(* Reference laser with X/Y motors (REFT): thin ND-framework state-mover
   wrapper. In/out mover via FB_PositionStatePMPSND, plus a tick site for
   the laser power/dimmer (FB_REF_Laser) and the X/Y motors. Caller-owned
   axes, stage/state arrays, fast-fault and arbiter injected via FB_Init
   REFERENCE TO and forwarded to fbStates; toggles re-forwarded each cycle. *)
{attribute 'call_after_init'}
FUNCTION_BLOCK FB_REFT
VAR_INPUT
    (* Device-specific state-enum bridges. Typed as E_EpicsInOut (UINT
       base) so the caller surface is enum-checked; the inline-init
       below binds them to FB_PositionStatePMPSND's REFERENCE TO UINT
       params via the shared UINT base. Callers drive moves with
       `fbREF.eEnumSet := E_EpicsInOut.OUT;` and read
       `fbREF.eEnumGet`. *)
    // Set this to a non-unknown value to request a new move.
    {attribute 'pytmc' := '
        pv: MMS:STATE:SET
        io: io
    '}
    eEnumSet : E_EpicsInOut;
    (* Run-time toggles forwarded into fbStates each cycle. PMPSND
       captures these by value in its own FB_Init, so the body
       re-writes fbStates.* every cycle to track live caller changes. *)
    fTermMax               : LREAL := 200;
END_VAR
VAR


    {attribute 'pytmc' := 'pv: LAS'}
    fbLaser : FB_REF_Laser;

    axisRefX : REFERENCE TO AXIS_REF;
    axisREFY : REFERENCE TO AXIS_REF;
     {attribute 'pytmc' := '
        pv: TST:Y
        io: io
        axis-link:
    '}
    fbMotorX : FB_MotionStageNC(
        AxisRef := axisRefX,
        iPersistentDataStorage := iPersistentDataStorage,
        sName := 'X'
    );
     {attribute 'pytmc' := '
        pv: TST:Y
        io: io
        axis-link:
    '}
    fbMotorY : FB_MotionStageNC(
        AxisRef := axisREFY,
        iPersistentDataStorage := iPersistentDataStorage,
        sName := 'Y'
    );

    iPersistentDataStorage : LCLS_Tc_DevAbs.I_PersistentDataStorage;
    aiMotionStage : ARRAY[1..MotionConstants.MAX_STATE_MOTORS] OF I_MotionStage := [fbMotorX, fbMotorY];

    astPositionState : REFERENCE TO ARRAY[1..MotionConstants.MAX_STATE_MOTORS]
                         OF ARRAY[1..GeneralConstants.MAX_STATES] OF ST_PositionState;

    {attribute 'no_copy'}
    fbFFHWO               : REFERENCE TO FB_HardwareFFOutput;
    {attribute 'no_copy'}
    fbArbiter             : REFERENCE TO FB_Arbiter;

    sDeviceName           : STRING;
    sTransitionKey        : STRING;
    bEnableMotion         : BOOL := TRUE;
    bEnableBeamParams     : BOOL;
    bEnablePositionLimits : BOOL;
    bReadDBNow            : BOOL;

    bFileReaderBusy       : REFERENCE TO BOOL;
    bFileReaderError      : REFERENCE TO BOOL;
    (* One configurator per REF state (OUT, IN). Writes the per-state
       sName and fDelta. Ticked cyclically in the body AFTER fbStates
       so its writes win over the template baseline FB_StateSetup
       applied via FB_CC_StatePMPSConfig *)
    afbStateDefaults : ARRAY[1..2] OF FB_CC_DeviceStateDefaults[
        (stPositionState := astPositionState[1][E_EpicsInOut.OUT],
         sName           := 'OUT',
         fDelta          := FDELTA_DEFAULT),
        (stPositionState := astPositionState[1][E_EpicsInOut.IN],
         sName           := 'IN',
         fDelta          := FDELTA_DEFAULT)
    ];
    {attribute 'pytmc' := 'pv: MMS'}
    fbStates : FB_PositionStatePMPSND(
        aiMotionStage         := aiMotionStage,
        astPositionState      := astPositionState,
        nActiveMotorCount     := 1,
        eEnumSet              := eEnumSet,
        eEnumGet              := eEnumGet,
        bEnableMotion         := bEnableMotion,
        eMotionRequestPolicy  := E_MotionRequestPolicy.INTERRUPT,
        bEnableBeamParams     := bEnableBeamParams,
        bEnablePositionLimits := bEnablePositionLimits,
        bReadDBNow            := bReadDBNow,
        bFileReaderBusy       := bFileReaderBusy,
        bFileReaderError      := bFileReaderError,
        fbFFHWO               := fbFFHWO,
        fbArbiter             := fbArbiter,
        sDeviceName           := sDeviceName,
        sTransitionKey        := sTransitionKey
    );
    i : UINT;
    bFirstScan: BOOL := TRUE;
END_VAR
VAR_OUTPUT
    // The current position state as an enum.
    {attribute 'pytmc' := '
        pv: MMS:STATE:GET
        io: i
    '}
     eEnumGet : E_EpicsInOut;
    // The PMPS database lookup associated with the current position state.
    stDbStateParams: ST_DbStateParams;
END_VAR
VAR CONSTANT
    (* REF-wide default tolerance for state in-position detection,
       applied per-state by afbStateDefaults. *)
    FDELTA_DEFAULT : LREAL := 2;
END_VAR

IF NOT __ISVALIDREF(astPositionState)
   OR NOT __ISVALIDREF(fbFFHWO)
   OR NOT __ISVALIDREF(fbArbiter) THEN
    RETURN;
END_IF

IF bFirstScan THEN
    FOR i := 1 TO MotionConstants.MAX_STATE_MOTORS DO
        aiMotionStage[i].SetModeEnableLimits(
            LimBackward    := TRUE,
            LimForward     := TRUE,
            HomeEnable     := FALSE,
            BrakeMode      := E_StageBrakeMode.IF_ENABLED,
            EnableMode     := E_StageEnableMode.DURING_MOTION,
            HomeMode       := E_EpicsHomeCmd.LOW_LIMIT,
            UserEnable     := TRUE,
            HardwareEnable := TRUE
        );
        aiMotionStage[i].SetVelocity(Velocity:=15.5);
        aiMotionStage[i].RestoreMotionParams:= FALSE;
    END_FOR
    bFirstScan := FALSE;
END_IF

fbStates(stDbStateParams=> stDbStateParams);

fbLaser(fTermMax := fTermMax);

fbMotorY();
fbMotorX();

(* Auto-fired after FB_Init. fbStates' inline-init ran first and
   forwarded nil refs, so this re-supplies the now-valid refs via
   fbStates.CallAfterInitStateMover / CallAfterInitPMPS and writes the
   per-state device defaults. *)
{attribute 'call_after_init'}
METHOD CallAfterInit
VAR
    i : UINT;
END_VAR
afbStateDefaults[1].CallAfterInit(
    stPositionState := THIS^.astPositionState[1][E_EpicsInOut.OUT]
);
afbStateDefaults[2].CallAfterInit(
    stPositionState := THIS^.astPositionState[1][E_EpicsInOut.IN]
);

THIS^.fbStates.CallAfterInitStateMover(
    aiMotionStage         := aiMotionStage,
    astPositionState      := astPositionState,
    nActiveMotorCount     := 1,
    eEnumSet              := eEnumSet,
    eEnumGet              := eEnumGet,
    bEnableMotion         := bEnableMotion,
    eMotionRequestPolicy  := E_MotionRequestPolicy.INTERRUPT,
);

THIS^.fbStates.CallAfterInitPMPS(
    aiMotionStage         := aiMotionStage,
    astPositionState      := astPositionState,
    bEnableBeamParams     := bEnableBeamParams,
    bEnablePositionLimits := bEnablePositionLimits,
    bReadDBNow            := bReadDBNow,
    bFileReaderBusy       := bFileReaderBusy,
    bFileReaderError      := bFileReaderError,
    fbFFHWO               := fbFFHWO,
    fbArbiter             := fbArbiter,
    sDeviceName           := sDeviceName,
    sTransitionKey        := sTransitionKey
);
END_METHOD

//FB_Init is always available implicitly and it is used primarily for initialization.
//The return value is not evaluated. For a specific influence, you can also declare the
//methods explicitly and provide additional code there with the standard initialization
//code. You can evaluate the return value.
METHOD FB_Init: BOOL
VAR_INPUT
    bInitRetains: BOOL; // TRUE: the retain variables are initialized (reset warm / reset cold)
    bInCopyCode: BOOL;  // TRUE: the instance will be copied to the copy code afterward (online change)
    astPositionState       : REFERENCE TO ARRAY[1..MotionConstants.MAX_STATE_MOTORS]
                                            OF ARRAY[1..GeneralConstants.MAX_STATES] OF ST_PositionState;
    axisRefX : REFERENCE TO AXIS_REF;
    axisREFY : REFERENCE TO AXIS_REF;
    fbFFHWO                : REFERENCE TO FB_HardwareFFOutput;
    fbArbiter              : REFERENCE TO FB_Arbiter;
    sDeviceName            : STRING;
    sTransitionKey         : STRING;
    bEnableBeamParams      : BOOL;
    bEnablePositionLimits  : BOOL;
    bReadDBNow             : BOOL;
    bFileReaderBusy       : REFERENCE TO BOOL;
    bFileReaderError      : REFERENCE TO BOOL;
END_VAR
THIS^.astPositionState REF= astPositionState;
THIS^.axisRefX REF= axisRefX;
THIS^.axisREFY REF= axisREFY;
THIS^.fbFFHWO          REF= fbFFHWO;
THIS^.fbArbiter        REF= fbArbiter;
THIS^.sDeviceName      := sDeviceName;
THIS^.sTransitionKey   := sTransitionKey;
THIS^.bEnableBeamParams    := bEnableBeamParams;
THIS^.bEnablePositionLimits:= bEnablePositionLimits;
THIS^.bReadDBNow           := bReadDBNow;
THIS^.bFileReaderBusy       REF= bFileReaderBusy;
THIS^.bFileReaderError      REF= bFileReaderError;
END_METHOD

PROPERTY MaintMode : BOOL
GET
MaintMode := fbStates.stPMPSEpicsToPlc.bMaintMode;
END_GET
SET
fbStates.stPMPSEpicsToPlc.bMaintMode := MaintMode;
END_SET
END_PROPERTY

END_FUNCTION_BLOCK

(* stored: Version 1.1.0.1
   POU FB_REFT: Id {47c5b9d9-9678-455e-bc10-47c8a3ff0d4d}, SpecialFunc None
   Method CallAfterInit: Id {63a790f3-6748-45a1-920d-20a6eea6f116}
   Method FB_Init: Id {301eb156-3f31-4082-918e-0cd66d16ae0e}
   Property MaintMode: Id {e812e1b4-de37-41cb-842e-47b8e1a6eceb}
   Get Get: Id {07a21e45-37ac-453c-b42c-f50717ec85f0}
   Set Set: Id {92f874b7-ba7a-4d08-a665-ff0140900579} *)
